GLOBALCONSTANTS SubStrings (* Global constants *)
  (* Standard: 61499-1 *)
  (* Version 1.0, 2026-09-11, Franz Höpfinger, Meisterschulen am Ostbahnhof *)
  PACKAGE Meins::InputOutputTester::Button_AI_Calibrate_3P_OPC_UA;
  VAR_GLOBAL CONSTANT
    AIC_I1_RAW_WRITE : WSTRING := "opc_ua[WRITE;/Objects/AnalogCalibrated/I1/RAW,1:s=AIC_I1_RAW]";
    AIC_I1_CAL_WRITE : WSTRING := "opc_ua[WRITE;/Objects/AnalogCalibrated/I1/CAL,1:s=AIC_I1_CAL]";
    AIC_I2_RAW_WRITE : WSTRING := "opc_ua[WRITE;/Objects/AnalogCalibrated/I2/RAW,1:s=AIC_I2_RAW]";
    AIC_I2_CAL_WRITE : WSTRING := "opc_ua[WRITE;/Objects/AnalogCalibrated/I2/CAL,1:s=AIC_I2_CAL]";
    AIC_I3_RAW_WRITE : WSTRING := "opc_ua[WRITE;/Objects/AnalogCalibrated/I3/RAW,1:s=AIC_I3_RAW]";
    AIC_I3_CAL_WRITE : WSTRING := "opc_ua[WRITE;/Objects/AnalogCalibrated/I3/CAL,1:s=AIC_I3_CAL]";
    AIC_I4_RAW_WRITE : WSTRING := "opc_ua[WRITE;/Objects/AnalogCalibrated/I4/RAW,1:s=AIC_I4_RAW]";
    AIC_I4_CAL_WRITE : WSTRING := "opc_ua[WRITE;/Objects/AnalogCalibrated/I4/CAL,1:s=AIC_I4_CAL]";
    AIC_I5_RAW_WRITE : WSTRING := "opc_ua[WRITE;/Objects/AnalogCalibrated/I5/RAW,1:s=AIC_I5_RAW]";
    AIC_I5_CAL_WRITE : WSTRING := "opc_ua[WRITE;/Objects/AnalogCalibrated/I5/CAL,1:s=AIC_I5_CAL]";
    AIC_I6_RAW_WRITE : WSTRING := "opc_ua[WRITE;/Objects/AnalogCalibrated/I6/RAW,1:s=AIC_I6_RAW]";
    AIC_I6_CAL_WRITE : WSTRING := "opc_ua[WRITE;/Objects/AnalogCalibrated/I6/CAL,1:s=AIC_I6_CAL]";
    AIC_I7_RAW_WRITE : WSTRING := "opc_ua[WRITE;/Objects/AnalogCalibrated/I7/RAW,1:s=AIC_I7_RAW]";
    AIC_I7_CAL_WRITE : WSTRING := "opc_ua[WRITE;/Objects/AnalogCalibrated/I7/CAL,1:s=AIC_I7_CAL]";
    AIC_I8_RAW_WRITE : WSTRING := "opc_ua[WRITE;/Objects/AnalogCalibrated/I8/RAW,1:s=AIC_I8_RAW]";
    AIC_I8_CAL_WRITE : WSTRING := "opc_ua[WRITE;/Objects/AnalogCalibrated/I8/CAL,1:s=AIC_I8_CAL]";
    AIC_I1_MIN_METHOD : WSTRING := "opc_ua[CREATE_METHOD;/Objects/AnalogCalibrated3P/I1/MINMethod,1:s=AIC_I1_MIN_METHOD]";
    AIC_I1_MID_METHOD : WSTRING := "opc_ua[CREATE_METHOD;/Objects/AnalogCalibrated3P/I1/MIDMethod,1:s=AIC_I1_MID_METHOD]";
    AIC_I1_MID_READ : WSTRING := "opc_ua[READ;/Objects/AnalogCalibrated/I1/MID,1:s=AIC_I1_MID]";
    AIC_I1_MAX_METHOD : WSTRING := "opc_ua[CREATE_METHOD;/Objects/AnalogCalibrated3P/I1/MAXMethod,1:s=AIC_I1_MAX_METHOD]";
    AIC_I2_MIN_METHOD : WSTRING := "opc_ua[CREATE_METHOD;/Objects/AnalogCalibrated3P/I2/MINMethod,1:s=AIC_I2_MIN_METHOD]";
    AIC_I2_MID_METHOD : WSTRING := "opc_ua[CREATE_METHOD;/Objects/AnalogCalibrated3P/I2/MIDMethod,1:s=AIC_I2_MID_METHOD]";
    AIC_I2_MID_READ : WSTRING := "opc_ua[READ;/Objects/AnalogCalibrated/I2/MID,1:s=AIC_I2_MID]";
    AIC_I2_MAX_METHOD : WSTRING := "opc_ua[CREATE_METHOD;/Objects/AnalogCalibrated3P/I2/MAXMethod,1:s=AIC_I2_MAX_METHOD]";
    AIC_I3_MIN_METHOD : WSTRING := "opc_ua[CREATE_METHOD;/Objects/AnalogCalibrated3P/I3/MINMethod,1:s=AIC_I3_MIN_METHOD]";
    AIC_I3_MID_METHOD : WSTRING := "opc_ua[CREATE_METHOD;/Objects/AnalogCalibrated3P/I3/MIDMethod,1:s=AIC_I3_MID_METHOD]";
    AIC_I3_MID_READ : WSTRING := "opc_ua[READ;/Objects/AnalogCalibrated/I3/MID,1:s=AIC_I3_MID]";
    AIC_I3_MAX_METHOD : WSTRING := "opc_ua[CREATE_METHOD;/Objects/AnalogCalibrated3P/I3/MAXMethod,1:s=AIC_I3_MAX_METHOD]";
    AIC_I4_MIN_METHOD : WSTRING := "opc_ua[CREATE_METHOD;/Objects/AnalogCalibrated3P/I4/MINMethod,1:s=AIC_I4_MIN_METHOD]";
    AIC_I4_MID_METHOD : WSTRING := "opc_ua[CREATE_METHOD;/Objects/AnalogCalibrated3P/I4/MIDMethod,1:s=AIC_I4_MID_METHOD]";
    AIC_I4_MID_READ : WSTRING := "opc_ua[READ;/Objects/AnalogCalibrated/I4/MID,1:s=AIC_I4_MID]";
    AIC_I4_MAX_METHOD : WSTRING := "opc_ua[CREATE_METHOD;/Objects/AnalogCalibrated3P/I4/MAXMethod,1:s=AIC_I4_MAX_METHOD]";
    AIC_I5_MIN_METHOD : WSTRING := "opc_ua[CREATE_METHOD;/Objects/AnalogCalibrated3P/I5/MINMethod,1:s=AIC_I5_MIN_METHOD]";
    AIC_I5_MID_METHOD : WSTRING := "opc_ua[CREATE_METHOD;/Objects/AnalogCalibrated3P/I5/MIDMethod,1:s=AIC_I5_MID_METHOD]";
    AIC_I5_MID_READ : WSTRING := "opc_ua[READ;/Objects/AnalogCalibrated/I5/MID,1:s=AIC_I5_MID]";
    AIC_I5_MAX_METHOD : WSTRING := "opc_ua[CREATE_METHOD;/Objects/AnalogCalibrated3P/I5/MAXMethod,1:s=AIC_I5_MAX_METHOD]";
    AIC_I6_MIN_METHOD : WSTRING := "opc_ua[CREATE_METHOD;/Objects/AnalogCalibrated3P/I6/MINMethod,1:s=AIC_I6_MIN_METHOD]";
    AIC_I6_MID_METHOD : WSTRING := "opc_ua[CREATE_METHOD;/Objects/AnalogCalibrated3P/I6/MIDMethod,1:s=AIC_I6_MID_METHOD]";
    AIC_I6_MID_READ : WSTRING := "opc_ua[READ;/Objects/AnalogCalibrated/I6/MID,1:s=AIC_I6_MID]";
    AIC_I6_MAX_METHOD : WSTRING := "opc_ua[CREATE_METHOD;/Objects/AnalogCalibrated3P/I6/MAXMethod,1:s=AIC_I6_MAX_METHOD]";
    AIC_I7_MIN_METHOD : WSTRING := "opc_ua[CREATE_METHOD;/Objects/AnalogCalibrated3P/I7/MINMethod,1:s=AIC_I7_MIN_METHOD]";
    AIC_I7_MID_METHOD : WSTRING := "opc_ua[CREATE_METHOD;/Objects/AnalogCalibrated3P/I7/MIDMethod,1:s=AIC_I7_MID_METHOD]";
    AIC_I7_MID_READ : WSTRING := "opc_ua[READ;/Objects/AnalogCalibrated/I7/MID,1:s=AIC_I7_MID]";
    AIC_I7_MAX_METHOD : WSTRING := "opc_ua[CREATE_METHOD;/Objects/AnalogCalibrated3P/I7/MAXMethod,1:s=AIC_I7_MAX_METHOD]";
    AIC_I8_MIN_METHOD : WSTRING := "opc_ua[CREATE_METHOD;/Objects/AnalogCalibrated3P/I8/MINMethod,1:s=AIC_I8_MIN_METHOD]";
    AIC_I8_MID_METHOD : WSTRING := "opc_ua[CREATE_METHOD;/Objects/AnalogCalibrated3P/I8/MIDMethod,1:s=AIC_I8_MID_METHOD]";
    AIC_I8_MID_READ : WSTRING := "opc_ua[READ;/Objects/AnalogCalibrated/I8/MID,1:s=AIC_I8_MID]";
    AIC_I8_MAX_METHOD : WSTRING := "opc_ua[CREATE_METHOD;/Objects/AnalogCalibrated3P/I8/MAXMethod,1:s=AIC_I8_MAX_METHOD]";
    Q01_READ : WSTRING := "opc_ua[READ;/Objects/DigitalOutput/Q01,1:s=Q01]";
    Q01_WRITE : WSTRING := "opc_ua[WRITE;/Objects/DigitalOutput/Q01,1:s=Q01]";
    Q02_READ : WSTRING := "opc_ua[READ;/Objects/DigitalOutput/Q02,1:s=Q02]";
    Q02_WRITE : WSTRING := "opc_ua[WRITE;/Objects/DigitalOutput/Q02,1:s=Q02]";
    Q03_READ : WSTRING := "opc_ua[READ;/Objects/DigitalOutput/Q03,1:s=Q03]";
    Q03_WRITE : WSTRING := "opc_ua[WRITE;/Objects/DigitalOutput/Q03,1:s=Q03]";
    Q04_READ : WSTRING := "opc_ua[READ;/Objects/DigitalOutput/Q04,1:s=Q04]";
    Q04_WRITE : WSTRING := "opc_ua[WRITE;/Objects/DigitalOutput/Q04,1:s=Q04]";
    Q05_READ : WSTRING := "opc_ua[READ;/Objects/DigitalOutput/Q05,1:s=Q05]";
    Q05_WRITE : WSTRING := "opc_ua[WRITE;/Objects/DigitalOutput/Q05,1:s=Q05]";
    Q06_READ : WSTRING := "opc_ua[READ;/Objects/DigitalOutput/Q06,1:s=Q06]";
    Q06_WRITE : WSTRING := "opc_ua[WRITE;/Objects/DigitalOutput/Q06,1:s=Q06]";
    Q07_READ : WSTRING := "opc_ua[READ;/Objects/DigitalOutput/Q07,1:s=Q07]";
    Q07_WRITE : WSTRING := "opc_ua[WRITE;/Objects/DigitalOutput/Q07,1:s=Q07]";
    Q08_READ : WSTRING := "opc_ua[READ;/Objects/DigitalOutput/Q08,1:s=Q08]";
    Q08_WRITE : WSTRING := "opc_ua[WRITE;/Objects/DigitalOutput/Q08,1:s=Q08]";
    Q09_READ : WSTRING := "opc_ua[READ;/Objects/DigitalOutput/Q09,1:s=Q09]";
    Q09_WRITE : WSTRING := "opc_ua[WRITE;/Objects/DigitalOutput/Q09,1:s=Q09]";
    Q10_READ : WSTRING := "opc_ua[READ;/Objects/DigitalOutput/Q10,1:s=Q10]";
    Q10_WRITE : WSTRING := "opc_ua[WRITE;/Objects/DigitalOutput/Q10,1:s=Q10]";
    Q11_READ : WSTRING := "opc_ua[READ;/Objects/DigitalOutput/Q11,1:s=Q11]";
    Q11_WRITE : WSTRING := "opc_ua[WRITE;/Objects/DigitalOutput/Q11,1:s=Q11]";
    Q12_READ : WSTRING := "opc_ua[READ;/Objects/DigitalOutput/Q12,1:s=Q12]";
    Q12_WRITE : WSTRING := "opc_ua[WRITE;/Objects/DigitalOutput/Q12,1:s=Q12]";
    Tick_WRITE : WSTRING := "opc_ua[WRITE;/Objects/System/Tick,1:s=System.Tick]";
    AIC_I1_MINREF_READ : WSTRING := "opc_ua[READ;/Objects/AnalogCalibrated/I1/MINREF,1:s=AIC_I1_MINREF]";
    AIC_I1_MINREF_WRITE : WSTRING := "opc_ua[WRITE;/Objects/AnalogCalibrated/I1/MINREF,1:s=AIC_I1_MINREF]";
    AIC_I1_MIDREF_READ : WSTRING := "opc_ua[READ;/Objects/AnalogCalibrated/I1/MIDREF,1:s=AIC_I1_MIDREF]";
    AIC_I1_MIDREF_WRITE : WSTRING := "opc_ua[WRITE;/Objects/AnalogCalibrated/I1/MIDREF,1:s=AIC_I1_MIDREF]";
    AIC_I1_MAXREF_READ : WSTRING := "opc_ua[READ;/Objects/AnalogCalibrated/I1/MAXREF,1:s=AIC_I1_MAXREF]";
    AIC_I1_MAXREF_WRITE : WSTRING := "opc_ua[WRITE;/Objects/AnalogCalibrated/I1/MAXREF,1:s=AIC_I1_MAXREF]";
    AIC_I2_MINREF_READ : WSTRING := "opc_ua[READ;/Objects/AnalogCalibrated/I2/MINREF,1:s=AIC_I2_MINREF]";
    AIC_I2_MINREF_WRITE : WSTRING := "opc_ua[WRITE;/Objects/AnalogCalibrated/I2/MINREF,1:s=AIC_I2_MINREF]";
    AIC_I2_MIDREF_READ : WSTRING := "opc_ua[READ;/Objects/AnalogCalibrated/I2/MIDREF,1:s=AIC_I2_MIDREF]";
    AIC_I2_MIDREF_WRITE : WSTRING := "opc_ua[WRITE;/Objects/AnalogCalibrated/I2/MIDREF,1:s=AIC_I2_MIDREF]";
    AIC_I2_MAXREF_READ : WSTRING := "opc_ua[READ;/Objects/AnalogCalibrated/I2/MAXREF,1:s=AIC_I2_MAXREF]";
    AIC_I2_MAXREF_WRITE : WSTRING := "opc_ua[WRITE;/Objects/AnalogCalibrated/I2/MAXREF,1:s=AIC_I2_MAXREF]";
    AIC_I3_MINREF_READ : WSTRING := "opc_ua[READ;/Objects/AnalogCalibrated/I3/MINREF,1:s=AIC_I3_MINREF]";
    AIC_I3_MINREF_WRITE : WSTRING := "opc_ua[WRITE;/Objects/AnalogCalibrated/I3/MINREF,1:s=AIC_I3_MINREF]";
    AIC_I3_MIDREF_READ : WSTRING := "opc_ua[READ;/Objects/AnalogCalibrated/I3/MIDREF,1:s=AIC_I3_MIDREF]";
    AIC_I3_MIDREF_WRITE : WSTRING := "opc_ua[WRITE;/Objects/AnalogCalibrated/I3/MIDREF,1:s=AIC_I3_MIDREF]";
    AIC_I3_MAXREF_READ : WSTRING := "opc_ua[READ;/Objects/AnalogCalibrated/I3/MAXREF,1:s=AIC_I3_MAXREF]";
    AIC_I3_MAXREF_WRITE : WSTRING := "opc_ua[WRITE;/Objects/AnalogCalibrated/I3/MAXREF,1:s=AIC_I3_MAXREF]";
    AIC_I4_MINREF_READ : WSTRING := "opc_ua[READ;/Objects/AnalogCalibrated/I4/MINREF,1:s=AIC_I4_MINREF]";
    AIC_I4_MINREF_WRITE : WSTRING := "opc_ua[WRITE;/Objects/AnalogCalibrated/I4/MINREF,1:s=AIC_I4_MINREF]";
    AIC_I4_MIDREF_READ : WSTRING := "opc_ua[READ;/Objects/AnalogCalibrated/I4/MIDREF,1:s=AIC_I4_MIDREF]";
    AIC_I4_MIDREF_WRITE : WSTRING := "opc_ua[WRITE;/Objects/AnalogCalibrated/I4/MIDREF,1:s=AIC_I4_MIDREF]";
    AIC_I4_MAXREF_READ : WSTRING := "opc_ua[READ;/Objects/AnalogCalibrated/I4/MAXREF,1:s=AIC_I4_MAXREF]";
    AIC_I4_MAXREF_WRITE : WSTRING := "opc_ua[WRITE;/Objects/AnalogCalibrated/I4/MAXREF,1:s=AIC_I4_MAXREF]";
    AIC_I5_MINREF_READ : WSTRING := "opc_ua[READ;/Objects/AnalogCalibrated/I5/MINREF,1:s=AIC_I5_MINREF]";
    AIC_I5_MINREF_WRITE : WSTRING := "opc_ua[WRITE;/Objects/AnalogCalibrated/I5/MINREF,1:s=AIC_I5_MINREF]";
    AIC_I5_MIDREF_READ : WSTRING := "opc_ua[READ;/Objects/AnalogCalibrated/I5/MIDREF,1:s=AIC_I5_MIDREF]";
    AIC_I5_MIDREF_WRITE : WSTRING := "opc_ua[WRITE;/Objects/AnalogCalibrated/I5/MIDREF,1:s=AIC_I5_MIDREF]";
    AIC_I5_MAXREF_READ : WSTRING := "opc_ua[READ;/Objects/AnalogCalibrated/I5/MAXREF,1:s=AIC_I5_MAXREF]";
    AIC_I5_MAXREF_WRITE : WSTRING := "opc_ua[WRITE;/Objects/AnalogCalibrated/I5/MAXREF,1:s=AIC_I5_MAXREF]";
    AIC_I6_MINREF_READ : WSTRING := "opc_ua[READ;/Objects/AnalogCalibrated/I6/MINREF,1:s=AIC_I6_MINREF]";
    AIC_I6_MINREF_WRITE : WSTRING := "opc_ua[WRITE;/Objects/AnalogCalibrated/I6/MINREF,1:s=AIC_I6_MINREF]";
    AIC_I6_MIDREF_READ : WSTRING := "opc_ua[READ;/Objects/AnalogCalibrated/I6/MIDREF,1:s=AIC_I6_MIDREF]";
    AIC_I6_MIDREF_WRITE : WSTRING := "opc_ua[WRITE;/Objects/AnalogCalibrated/I6/MIDREF,1:s=AIC_I6_MIDREF]";
    AIC_I6_MAXREF_READ : WSTRING := "opc_ua[READ;/Objects/AnalogCalibrated/I6/MAXREF,1:s=AIC_I6_MAXREF]";
    AIC_I6_MAXREF_WRITE : WSTRING := "opc_ua[WRITE;/Objects/AnalogCalibrated/I6/MAXREF,1:s=AIC_I6_MAXREF]";
    AIC_I7_MINREF_READ : WSTRING := "opc_ua[READ;/Objects/AnalogCalibrated/I7/MINREF,1:s=AIC_I7_MINREF]";
    AIC_I7_MINREF_WRITE : WSTRING := "opc_ua[WRITE;/Objects/AnalogCalibrated/I7/MINREF,1:s=AIC_I7_MINREF]";
    AIC_I7_MIDREF_READ : WSTRING := "opc_ua[READ;/Objects/AnalogCalibrated/I7/MIDREF,1:s=AIC_I7_MIDREF]";
    AIC_I7_MIDREF_WRITE : WSTRING := "opc_ua[WRITE;/Objects/AnalogCalibrated/I7/MIDREF,1:s=AIC_I7_MIDREF]";
    AIC_I7_MAXREF_READ : WSTRING := "opc_ua[READ;/Objects/AnalogCalibrated/I7/MAXREF,1:s=AIC_I7_MAXREF]";
    AIC_I7_MAXREF_WRITE : WSTRING := "opc_ua[WRITE;/Objects/AnalogCalibrated/I7/MAXREF,1:s=AIC_I7_MAXREF]";
    AIC_I8_MINREF_READ : WSTRING := "opc_ua[READ;/Objects/AnalogCalibrated/I8/MINREF,1:s=AIC_I8_MINREF]";
    AIC_I8_MINREF_WRITE : WSTRING := "opc_ua[WRITE;/Objects/AnalogCalibrated/I8/MINREF,1:s=AIC_I8_MINREF]";
    AIC_I8_MIDREF_READ : WSTRING := "opc_ua[READ;/Objects/AnalogCalibrated/I8/MIDREF,1:s=AIC_I8_MIDREF]";
    AIC_I8_MIDREF_WRITE : WSTRING := "opc_ua[WRITE;/Objects/AnalogCalibrated/I8/MIDREF,1:s=AIC_I8_MIDREF]";
    AIC_I8_MAXREF_READ : WSTRING := "opc_ua[READ;/Objects/AnalogCalibrated/I8/MAXREF,1:s=AIC_I8_MAXREF]";
    AIC_I8_MAXREF_WRITE : WSTRING := "opc_ua[WRITE;/Objects/AnalogCalibrated/I8/MAXREF,1:s=AIC_I8_MAXREF]";
  END_VAR
END_GLOBALCONSTANTS
